# EPICS alarm handler configuration: test.win32.alhConfig
$BEEPSEVERITY  MAJOR
GROUP    NULL   JBATestMainGroup
$COMMAND command /K dir
$GUIDANCE
This is the text guidance for JBATestMainGroup alarms.
This is more guidance for JBATestMainGroup alarms.
$END
CHANNEL  JBATestMainGroup  jba:Example1 -----
CHANNEL  JBATestMainGroup  jba:Example2 -----
GROUP JBATestMainGroup  Group1
$GUIDANCE
This is the text guidance for group Group1.
This is more guidance for group Group1.
$END
$COMMAND start probe.exe
CHANNEL  Group1  jba:Example3 -----
CHANNEL  Group1  jba:Example4 -----
GROUP    Group1   Group1.SubGroup1
$GUIDANCE
This is the text guidance for Group1.SubGroup1.
This is more guidance for Group1.SubGroup1.
$END
CHANNEL  Group1.SubGroup1  jba:Example5 -----
CHANNEL  Group1.SubGroup1  jba:Example6 -----
GROUP    Group1.SubGroup1  Group1.SubSubGroup1
CHANNEL  Group1.SubSubGroup1  jba:Example11 -----
CHANNEL  Group1.SubSubGroup1  jba:Example12 -----
GROUP    Group1.SubGroup1  Group1.SubSubGroup2
CHANNEL  Group1.SubSubGroup2  jba:Example13 -----
CHANNEL  Group1.SubSubGroup2  jba:Example14 -----
GROUP    Group1   Group1.SubGroup2
$GUIDANCE
This is the text guidance for Group1.SubGroup2.
This is more guidance for Group1.SubGroup2.
$END
CHANNEL  Group1.SubGroup2  jba:Example7 -----
CHANNEL  Group1.SubGroup2  jba:Example8 -----
GROUP JBATestMainGroup  Group2
$ALIAS   AliasForGroup2
CHANNEL  Group2  jba:Example9 -----
CHANNEL  Group2  jba:Example10 -----
GROUP  JBATestMainGroup EvansGroup
CHANNEL  EvansGroup  evans:calc
CHANNEL  EvansGroup  evans:bo01
CHANNEL  EvansGroup  Xorbit:S1A:H1:CurrentAO
